# EPICS autosave request: GalilSup/Db/GALIL_controller_settings.req
# based on iocBoot/iocGalilTest/GalilTest_DMC01Settings.req

# scan and SaveData settings
file standardScans_settings.req P=$(P)DMC$(CCP):
file saveData_settings.req P=$(P)DMC$(CCP):

# Controller settings that motorRecord does not support
file "galil_dmc_ctrl.req" P=$(P)DMC$(CCP):

# User array names
file "galil_user_array.req" P=$(P)DMC$(CCP):

# Motor record settings
# Real motors
file "motor_settings.req" P=$(P), M=MTR$(CCP)01
file "motor_settings.req" P=$(P), M=MTR$(CCP)02
file "motor_settings.req" P=$(P), M=MTR$(CCP)03
file "motor_settings.req" P=$(P), M=MTR$(CCP)04
file "motor_settings.req" P=$(P), M=MTR$(CCP)05
file "motor_settings.req" P=$(P), M=MTR$(CCP)06
file "motor_settings.req" P=$(P), M=MTR$(CCP)07
file "motor_settings.req" P=$(P), M=MTR$(CCP)08

# Motor record settings not included in community req file
# Real motors
file "galil_motor_settings.req" P=$(P), M=MTR$(CCP)01
file "galil_motor_settings.req" P=$(P), M=MTR$(CCP)02
file "galil_motor_settings.req" P=$(P), M=MTR$(CCP)03
file "galil_motor_settings.req" P=$(P), M=MTR$(CCP)04
file "galil_motor_settings.req" P=$(P), M=MTR$(CCP)05
file "galil_motor_settings.req" P=$(P), M=MTR$(CCP)06
file "galil_motor_settings.req" P=$(P), M=MTR$(CCP)07
file "galil_motor_settings.req" P=$(P), M=MTR$(CCP)08

# Motor settings that motorRecord does not support
# Real motors only
file "galil_motor_extras.req" P=$(P), M=MTR$(CCP)01
file "galil_motor_extras.req" P=$(P), M=MTR$(CCP)02
file "galil_motor_extras.req" P=$(P), M=MTR$(CCP)03
file "galil_motor_extras.req" P=$(P), M=MTR$(CCP)04
file "galil_motor_extras.req" P=$(P), M=MTR$(CCP)05
file "galil_motor_extras.req" P=$(P), M=MTR$(CCP)06
file "galil_motor_extras.req" P=$(P), M=MTR$(CCP)07
file "galil_motor_extras.req" P=$(P), M=MTR$(CCP)08

# Motor record settings
# Coordinate system (cs) motors
file "motor_settings.req" P=$(P), M=MTR$(CCP)09
file "motor_settings.req" P=$(P), M=MTR$(CCP)10
file "motor_settings.req" P=$(P), M=MTR$(CCP)11
file "motor_settings.req" P=$(P), M=MTR$(CCP)12
file "motor_settings.req" P=$(P), M=MTR$(CCP)13
file "motor_settings.req" P=$(P), M=MTR$(CCP)14
file "motor_settings.req" P=$(P), M=MTR$(CCP)15
file "motor_settings.req" P=$(P), M=MTR$(CCP)16

# Motor record settings not included in community req file
# Coordinate system (cs) motors
file "galil_motor_settings.req" P=$(P), M=MTR$(CCP)09
file "galil_motor_settings.req" P=$(P), M=MTR$(CCP)10
file "galil_motor_settings.req" P=$(P), M=MTR$(CCP)11
file "galil_motor_settings.req" P=$(P), M=MTR$(CCP)12
file "galil_motor_settings.req" P=$(P), M=MTR$(CCP)13
file "galil_motor_settings.req" P=$(P), M=MTR$(CCP)14
file "galil_motor_settings.req" P=$(P), M=MTR$(CCP)15
file "galil_motor_settings.req" P=$(P), M=MTR$(CCP)16

# Digital inputs
#file "galil_digital_in_bit.req" P=DMC$(CCP):, R=Galil0Bi0

# Digital Outputs
#file "galil_digital_out_bit.req" P=DMC$(CCP):, R=Galil0Bo0

# Analogue inputs
#file "galil_analog_in.req" P=DMC$(CCP):, R=GalilAi0

# Analogue outputs
#file "galil_analog_out.req" P=DMC$(CCP):, R=GalilAo0

# galil userdef records
file "galil_userdef_records8.req" P=$(P), M=MTR$(CCP), GS=K1
file "galil_userdef_records8.req" P=$(P), M=MTR$(CCP), GS=K2
file "galil_userdef_records8.req" P=$(P), M=MTR$(CCP), GS=K3
file "galil_userdef_records8.req" P=$(P), M=MTR$(CCP), GS=IL
file "galil_userdef_records8.req" P=$(P), M=MTR$(CCP), GS=FV
file "galil_userdef_records8.req" P=$(P), M=MTR$(CCP), GS=FC
file "galil_userdef_records8.req" P=$(P), M=MTR$(CCP), GS=FA
file "galil_userdef_records8.req" P=$(P), M=MTR$(CCP), GS=FN
file "galil_userdef_records8.req" P=$(P), M=MTR$(CCP), GS=ZP
file "galil_userdef_records8.req" P=$(P), M=MTR$(CCP), GS=ZN
file "galil_userdef_records8.req" P=$(P), M=MTR$(CCP), GS=TL
file "galil_userdef_records8.req" P=$(P), M=MTR$(CCP), GS=CP
file "galil_userdef_records8.req" P=$(P), M=MTR$(CCP), GS=CT
file "galil_userdef_records8.req" P=$(P), M=MTR$(CCP), GS=AF
